KUKA KRL program: Zero_Position.src, Zero_Position.dat

--- Zero_Position.src ---
&ACCESS RVP
&REL 1
&COMMENT Kiem tra vi tri zero
DEF Zero_Position()
  ;FOLD INI
    ;FOLD BASISTECH INI
      BAS(#INITMOV, 0)
    ;ENDFOLD
  ;ENDFOLD

  ; Di chuyen tat ca truc ve 0 do
  PTP {A1 0, A2 0, A3 0, A4 0, A5 0, A6 0} Vel=10% DEFAULT

  HALT

  PTP HOME Vel=100% DEFAULT

END

--- Zero_Position.dat ---
&ACCESS RV
&REL 1
DEFDAT Zero_Position PUBLIC
  DECL E6POS HOME={A1 0.0, A2 -90.0, A3 90.0, A4 0.0, A5 0.0, A6 0.0}
ENDDAT
